(* Schneider Machine Expert - Basic project Test_Pump, file version 3.0.0.0 *)
(* ProjectInformations: Name=Test_Pump *)

HARDWARE
  Cpu 0: TM221CE24T
  ModuleExtensionObject 0: TM3AI4/G
  EthernetConfiguration: NetworkName=M221, IpAllocationMode=ByDhcp, IpAddress=192.168.1.10, SubnetMask=255.255.255.0
  SerialLineConfiguration: Baud=Baud19200, Parity=ParityEven, DataBits=DataBits8, StopBits=StopBits1, PhysicalMedium=PhysicalMediumRs485, TransmissionMode=TransmissionModeModbusRtu, SlaveId=1, Addressing=SlaveAddressing
  MastTask: UsePeriodScanMode=false, PeriodScan=100
  FastTask: Period=255
  CpuBehavior: StartingMode=StartAsPreviousState, AutoSaveRamOnEeprom=true, WatchdogPeriod=250

SYMBOLS  (address, symbol, comment, settings)
  %M0       PUMP_RUN  "Pump Running Status"
  %M1       PRES_LOW  "Pressure Below Low Setpoint"
  %M2       PRES_HIGH  "Pressure Above High Setpoint"
  %M3       AUTO_CMD  "Auto Mode Pump Command"
  %M4       MAN_START  "Manual Start Command"
  %M5       AUTO_START  "Auto Start Command"
  %I0.0     PB_START
  %I0.1     PB_STOP
  %I0.2     ESTOP
  %I0.3     SS_AUTO
  %Q0.0     PUMP_OUT
  %Q0.1     LT_RUN
  %Q0.2     LT_AUTO
  %Q0.3     LT_PRES_HI
  %IW1.0    PRES_AIN  [Type=Type_4_20mA, Scope=Scope_Customized, Minimum=0, Maximum=10000]

POU Test_Pump
  (* SectionNumber=1 *)

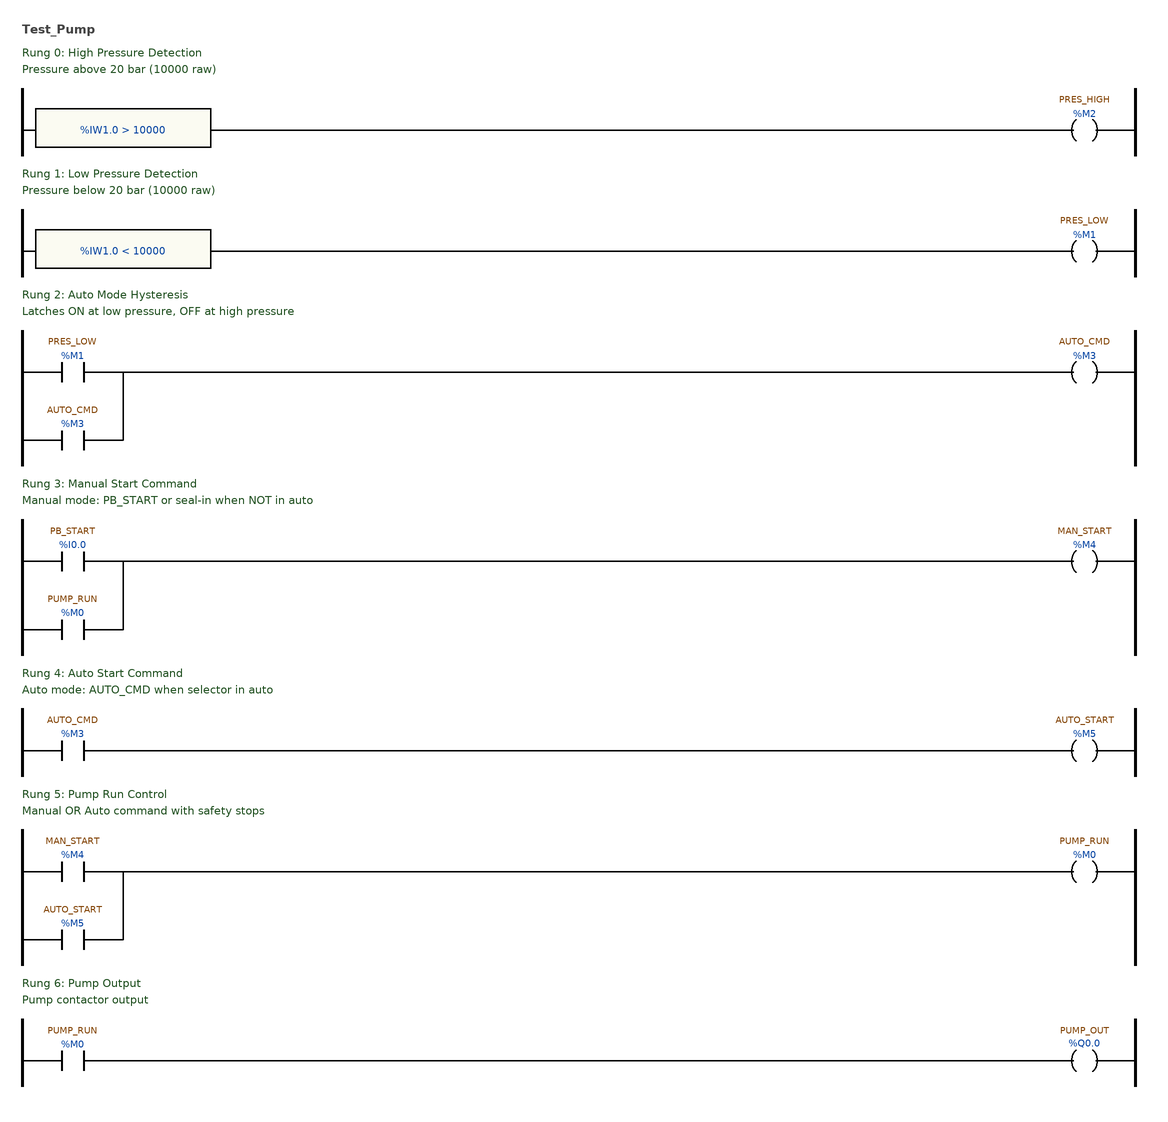

// Rung 0: High Pressure Detection
// Pressure above 20 bar (10000 raw)
  LD [ %IW1.0 > 10000 ]   (* PRES_AIN *)
  ST %M2                  (* PRES_HIGH *)
  // as ST:
  //   PRES_HIGH := PRES_AIN > 10000;

// Rung 1: Low Pressure Detection
// Pressure below 20 bar (10000 raw)
  LD [ %IW1.0 < 10000 ]   (* PRES_AIN *)
  ST %M1                  (* PRES_LOW *)
  // as ST:
  //   PRES_LOW := PRES_AIN < 10000;

// Rung 2: Auto Mode Hysteresis
// Latches ON at low pressure, OFF at high pressure
  LD %M1                  (* PRES_LOW *)
  OR %M3                  (* AUTO_CMD *)
  ST %M3                  (* AUTO_CMD *)
  // as ST:
  //   AUTO_CMD := PRES_LOW OR AUTO_CMD;

// Rung 3: Manual Start Command
// Manual mode: PB_START or seal-in when NOT in auto
  LD %I0.0                (* PB_START *)
  OR %M0                  (* PUMP_RUN *)
  ST %M4                  (* MAN_START *)
  // as ST:
  //   MAN_START := PB_START OR PUMP_RUN;

// Rung 4: Auto Start Command
// Auto mode: AUTO_CMD when selector in auto
  LD %M3                  (* AUTO_CMD *)
  ST %M5                  (* AUTO_START *)
  // as ST:
  //   AUTO_START := AUTO_CMD;

// Rung 5: Pump Run Control
// Manual OR Auto command with safety stops
  LD %M4                  (* MAN_START *)
  OR %M5                  (* AUTO_START *)
  ST %M0                  (* PUMP_RUN *)
  // as ST:
  //   PUMP_RUN := MAN_START OR AUTO_START;

// Rung 6: Pump Output
// Pump contactor output
  LD %M0                  (* PUMP_RUN *)
  ST %Q0.0                (* PUMP_OUT *)
  // as ST:
  //   PUMP_OUT := PUMP_RUN;

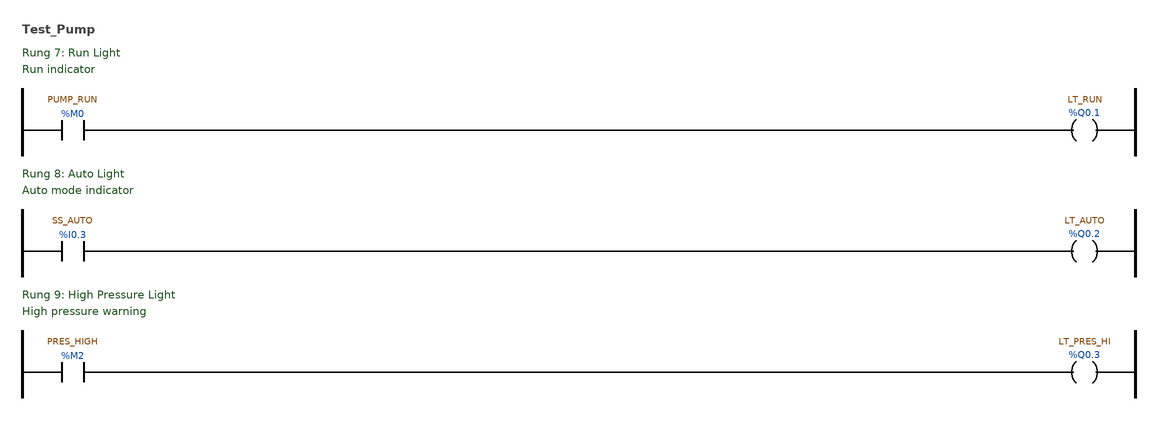

// Rung 7: Run Light
// Run indicator
  LD %M0                  (* PUMP_RUN *)
  ST %Q0.1                (* LT_RUN *)
  // as ST:
  //   LT_RUN := PUMP_RUN;

// Rung 8: Auto Light
// Auto mode indicator
  LD %I0.3                (* SS_AUTO *)
  ST %Q0.2                (* LT_AUTO *)
  // as ST:
  //   LT_AUTO := SS_AUTO;

// Rung 9: High Pressure Light
// High pressure warning
  LD %M2                  (* PRES_HIGH *)
  ST %Q0.3                (* LT_PRES_HI *)
  // as ST:
  //   LT_PRES_HI := PRES_HIGH;
